TYPE (* EventFilter type used to subsribe/unsubscribe to/from the EventHandler *)
  (* Standard: 61499-2; Description: Copyright (c) 2019 fortiss GmbH This program and the accompanying materials are made available under the terms of the Eclipse Public License 2.0 which is available at https://www.eclipse.org/legal/epl-2.0/ SPDX-License-Identifier: EPL-2.0 *)
  (* Version 1.0, 2019-09-17, Jose Cabral, fortiss GmbH *)
  (* ASN.1 tag APPLICATION 1 *)
  EventFilter : STRUCT
    eventType : WSTRING; (* Event type, similar to topics in MQTT. *)
    consumer : ArrowheadSystem; (* The Subscriber ArrowheadSystem, that will consume the new events. *)
    sources : ARRAY [0..9] OF ArrowheadSystem; (* List of ArrowheadSystem the Subscriber wants to receive events from. *)
    startDate : DATE_AND_TIME; (* If set, the Subscriber wants to receive events with timestamps after this date-time. *)
    endDate : DATE_AND_TIME; (* If set, the Subscriber wants to receive events with timestamps before this date-time. *)
    filterMetadata : ARRAY [0..9] OF WSTRING; (* Metadata about the events, which can be used for further filtering. *)
    notifyUri : WSTRING; (* The URL subpath where the Event Handler should sent the new events to. *)
    matchMetadata : BOOL; (* Should the Event Handler filter events based on the metadata. *)
  END_STRUCT;
END_TYPE
